// TIA Portal V20 export
VAR_GLOBAL   // PLC tag table "LGR_Const_Equip_Status"
END_VAR
VAR_GLOBAL CONSTANT   // user constants
   STAT_NORMAL : Byte := 2#0000_0001;   // .X0
   STAT_IDLE : Byte := 2#0000_0010;   // .X1
   STAT_BUSY : Byte := 2#0000_0100;   // .X2
   STAT_ONLINE : Byte := 2#1000_0000;   // .X7
   STAT_FAULT : Byte := 2#0100_0000;   // .X6
END_VAR
